KUKA KRL program: main.src, main.dat

--- main.src ---
&ACCESS RVP
&REL 5
&COMMENT Main Program Demo
DEF main()
  ; --- 1. DEMO: System Initialization ---
  ; Notice Inlay Hint for BASE_DATA[1] and TOOL_DATA[1]
  $BASE = BASE_DATA[1]
  $TOOL = TOOL_DATA[1]

  $VEL.CP = 1.5
  $ACC.CP = 2.0

  PTP {A1 0, A2 -90, A3 90, A4 0, A5 30, A6 0}

  ; --- 2. DEMO: Signal Operations (Inlay Hints active here) ---
  ; Write "$OUT[4] = TRUE" or "$IN[1]" to see instant hints
  WAIT FOR $IN[1]  ; <- Will show diPartReady

  $OUT[4] = TRUE   ; <- Will show doGripperOpen
  $OUT[5] = FALSE  ; <- Will show doGripperClose

  ; Call subroutine
  executeProcessCycle()


  $OUT[10] = TRUE  ; <- Will show doCycleComplete
END

DEF executeProcessCycle()
  $TOOL = TOOL_DATA[1]
  $BASE = BASE_DATA[1]
  ; Basic sequence
  LIN {X 1200, Y -450, Z 950}
  WAIT SEC 0.5
  LIN {X 1200, Y -450, Z 800}
  $OUT[4] = FALSE
  $OUT[5] = TRUE
  WAIT SEC 1.0
END

--- main.dat ---
&ACCESS RVP
&REL 5
&COMMENT Main Program Data
DEFDAT main
  ; --- Local Point Declarations for Go-to-Definition & Diff ---
  DECL E6POS P1={X 1200.5, Y -450.0, Z 950.0, A 0.0, B 90.0, C 0.0, S 2, T 35}
  DECL E6POS P2={X 1200.5, Y -450.0, Z 800.0, A 0.0, B 90.0, C 0.0, S 2, T 35}
  DECL E6POS PICK_POINT={X 1450.0, Y 300.0, Z 650.0, A 45.0, B 0.0, C 180.0, S 6, T 19}
  DECL E6POS PLACE_POINT={X 1800.0, Y -200.0, Z 500.0, A -90.0, B 0.0, C 180.0, S 6, T 19}

  ; --- Local Motion Parameters ---
  DECL FDAT F1={TOOL_NO 1, BASE_NO 1, IPO_FRAME #BASE}
  DECL FDAT F2={TOOL_NO 1, BASE_NO 1, IPO_FRAME #BASE}
  DECL LDAT LPDAT1={VEL 2.0, ACC 100.0, APO_DIST 100.0, APO_FAC 50.0, AXIS_VEL 100.0, AXIS_ACC 100.0}
  DECL PDAT PPDAT1={VEL 100.0, ACC 100.0, APO_DIST 50.0}
ENDDAT
